TYPE tDataFrame_1 :
ARRAY[0..64] OF BYTE; // Normal Mode datagram
END_TYPE

(* stored: Version 1.1.0.1, ProductVersion 3.1.4024.9
   DUT tDataFrame_1: Id {f65a77b4-58bb-4f6d-a5c2-95c37e524a6e} *)
